INTERFACE ITestEventHandler_UsesEventArgs EXTENDS IEventHandlerBase

METHOD OnThisEvent
VAR_INPUT
    EventArgs : IStreamReader;
END_VAR
END_METHOD

END_INTERFACE

(* stored: Version 1.1.0.1, ProductVersion 3.1.4024.3
   Itf ITestEventHandler_UsesEventArgs: Id {dc6397c7-f4e5-4f33-835a-bf5aa350e6b7}
   Method OnThisEvent: Id {eb402ea7-bd0c-4a40-b0b1-133ce76d3ba0} *)
